SYSTEM TEST_CSW (* Test CLIENTW/SERVERW Configuration *)
  (* Standard: 61499-1 *)
  (* Version 0.0, 2004-10-19, JHC, Rockwell Automation *)
  DEVICE CLIENT : FRAME_DEVICE(BOUNDS := [100,100,150,125])
    RESOURCE RES1 : PANEL_RESOURCE(ROWS := 3, COLS := 1)
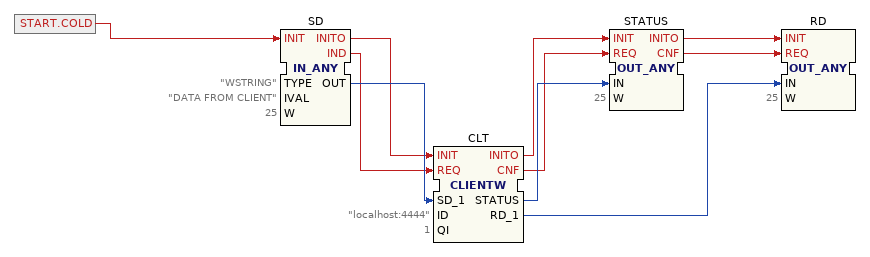
      FBS
        SD : IN_ANY(TYPE := "WSTRING", IVAL := "DATA FROM CLIENT", W := 25);
        CLT : CLIENTW(ID := "localhost:4444", QI := 1);
        STATUS : OUT_ANY(W := 25);
        RD : OUT_ANY(W := 25);
      END_FBS
      EVENT_CONNECTIONS
        START.COLD TO SD.INIT;
        SD.INITO TO CLT.INIT;
        SD.IND TO CLT.REQ;
        CLT.INITO TO STATUS.INIT;
        CLT.CNF TO STATUS.REQ;
        STATUS.INITO TO RD.INIT;
        STATUS.CNF TO RD.REQ;
      END_CONNECTIONS
      DATA_CONNECTIONS
        SD.OUT TO CLT.SD_1;
        CLT.STATUS TO STATUS.IN;
        CLT.RD_1 TO RD.IN;
      END_CONNECTIONS
    END_RESOURCE
  END_DEVICE
  DEVICE SERVER : FRAME_DEVICE(BOUNDS := [250,100,150,125])
    RESOURCE RES1 : PANEL_RESOURCE(ROWS := 3, COLS := 1)
      FBS
        SD : IN_ANY(TYPE := "WSTRING", IVAL := "DATA", W := 25);
        CLT : SERVERW(QI := 1, ID := "localhost:4444");
        STATUS : OUT_ANY(W := 25);
        RD : OUT_ANY(W := 25);
        CONC : FB_CONCAT(IN2 := " FROM SERVER"); (* Force WSTRING output to replace CLT.SD *)
      END_FBS
      EVENT_CONNECTIONS
        START.COLD TO SD.INIT;
        SD.INITO TO CLT.INIT;
        CLT.INITO TO STATUS.INIT;
        STATUS.INITO TO RD.INIT;
        STATUS.CNF TO RD.REQ;
        CLT.IND TO STATUS.REQ;
        SD.IND TO CONC.REQ;
        CONC.CNF TO CLT.RSP;
      END_CONNECTIONS
      DATA_CONNECTIONS
        CLT.STATUS TO STATUS.IN;
        CLT.RD_1 TO RD.IN;
        SD.OUT TO CONC.IN1;
        CONC.OUT TO CLT.SD_1;
      END_CONNECTIONS
    END_RESOURCE
  END_DEVICE
END_SYSTEM
